ABB RobotStudio station: Escalera.rspag

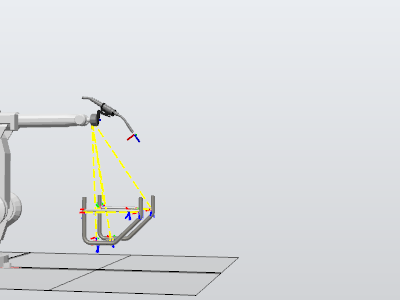
--- station ---
Station Project4 (saved by RobotStudio 23.2.10395.0)
Controller IRB1410_5_144
  mechanical unit ROB_1: IRB1410_5_144__01, 6 joints, base frame (0, 0, 0) mm
Layout (positions relative to the parent item):
  - IRB1410_5_144__01 [mechanism, from %ABB.RobotStudio.Models.IRB1410%\IRB1410_5_144_G_01.rslib] at (0, 0, 0) mm; joint values [0, 0, 0, 0, 0, 0] (rad or m)
  - AW_Gun_PSF_25 [mechanism, from %ABB.RobotStudio.Models.ArcWelding%\AW_Gun_PSF_25.rslib] at (955, 0, 1195) mm, rotated rx 0 ry 90 rz 0 deg
  - escalera [graphiccomponentgroup] at (1200, -200, 400) mm, rotated rx -90 ry 0 rz 0 deg
    - patasescalera:1 [part] at (-235.15, -185.03, 0) mm, size 475.4 x 362.7 x 25.4 mm
    - tubolargo:1 [part] at (-229.58, -85.03, -0.64) mm, rotated rx 90 ry 0 rz 0 deg, size 440 x 19 x 19 mm
    - patasescalera:2 [part] at (-235.69, -185.03, 370) mm, size 475.4 x 362.7 x 25.4 mm
    - tubolargo:2 [part] at (-231.19, -85.03, 370) mm, rotated rx 90 ry 0 rz 0 deg, size 440 x 19 x 19 mm
    - tubo peque\X\F1o:1 [part] at (123.63, -81.8, 370.84) mm, rotated rx -90 ry 89.5 rz -90 deg, size 370 x 19 x 19 mm
    - tubo peque\X\F1o:2 [part] at (-121.37, 167.61, 371.49) mm, rotated rx -90 ry 89.59 rz -90 deg, size 370 x 19 x 19 mm
Attachment: AW_Gun_PSF_25 is attached to IRB1410_5_144__01 / Link6
Targets, tools, work objects and paths stored in the station and not in the controller backup, written as RAPID:
! task T_ROB1
MODULE CalibData
  PERS tooldata AW_Gun:=[TRUE,[[119.5,0,352],[0.890213743,0,0.455543074,0]],[1,[0,0,100],[1,0,0,0],0,0,0]];
  TASK PERS wobjdata Workobject_1:=[FALSE,TRUE,"",[[0,0,0],[1,0,0,0]],[[0,0,0],[1,0,0,0]]];
ENDMODULE

! task T_ROB1
MODULE Module1
  CONST jointtarget Home:=[[0,0,0,0,0,0],[9E+09,9E+09,9E+09,9E+09,9E+09,9E+09]];
  CONST robtarget Mitad1:=[[976.781186414,170.702276534,494.530253281],[0.305176705,0.666129903,-0.637918703,-0.237060876],[-1,0,-1,0],[9E+09,9E+09,9E+09,9E+09,9E+09,9E+09]];
  CONST robtarget Inicio1:=[[972.88593197,180.494399691,477.051816875],[0.385830495,0.691371329,-0.592631267,-0.148083408],[-1,0,-1,0],[9E+09,9E+09,9E+09,9E+09,9E+09,9E+09]];
  CONST robtarget Fin1:=[[973.255,150,480],[0.037823374,0.524703407,-0.706148979,-0.473929685],[-1,0,-2,0],[9E+09,9E+09,9E+09,9E+09,9E+09,9E+09]];
  CONST robtarget Mitad2:=[[978.420658892,-200.453702036,494.554289293],[0.153565718,0.360544064,-0.853445443,-0.343593399],[-1,0,-1,0],[9E+09,9E+09,9E+09,9E+09,9E+09,9E+09]];
  CONST robtarget Fin2:=[[978.421,-220,470],[0.156146418,0.366952713,-0.850711042,-0.342424773],[-1,0,-1,0],[9E+09,9E+09,9E+09,9E+09,9E+09,9E+09]];
  CONST robtarget Inicio2:=[[978.421,-180,470],[0.158675671,0.365866136,-0.848327112,-0.348288837],[-1,0,-1,0],[9E+09,9E+09,9E+09,9E+09,9E+09,9E+09]];
  CONST robtarget Inicio3:=[[1400,-212.929,477.071],[0.120590477,-0.049950211,0.915975615,0.379409523],[-1,-1,1,0],[9E+09,9E+09,9E+09,9E+09,9E+09,9E+09]];
  CONST robtarget Mitad3:=[[1400,-200,490],[0.130526192,0,0.991444861,0],[-1,-1,0,0],[9E+09,9E+09,9E+09,9E+09,9E+09,9E+09]];
  CONST robtarget Fin3:=[[1400,-187.071,477.071],[0.120590477,0.049950211,0.915975615,-0.379409523],[0,0,-1,0],[9E+09,9E+09,9E+09,9E+09,9E+09,9E+09]];
  CONST robtarget Inicio4:=[[1333.134,-191.144,484.911],[0.254887002,0.044943456,-0.951251243,0.167731259],[-1,0,-1,0],[9E+09,9E+09,9E+09,9E+09,9E+09,9E+09]];
  CONST robtarget Mitad4:=[[1323,-191.144,484.911],[0,0,1,0],[-1,0,-1,0],[9E+09,9E+09,9E+09,9E+09,9E+09,9E+09]];
  CONST robtarget Fin4:=[[1313,-191.144,484.911],[0.130526192,0,0.991444861,0],[-1,1,-2,0],[9E+09,9E+09,9E+09,9E+09,9E+09,9E+09]];
  CONST robtarget Inicio5:=[[1313,153.856,484.911],[0.130526192,0,0.991444861,0],[0,0,-1,0],[9E+09,9E+09,9E+09,9E+09,9E+09,9E+09]];
  CONST robtarget Mitad5:=[[1323,160,484.911],[0,0,1,0],[0,1,-2,0],[9E+09,9E+09,9E+09,9E+09,9E+09,9E+09]];
  CONST robtarget Fin5:=[[1333,153.856,480],[0,0,1,0],[0,1,-2,0],[9E+09,9E+09,9E+09,9E+09,9E+09,9E+09]];
  CONST robtarget Inicio6:=[[1405,157.392,476.464],[0.128543206,-0.022665635,0.976382586,0.172162593],[-1,-1,1,0],[9E+09,9E+09,9E+09,9E+09,9E+09,9E+09]];
  CONST robtarget Mitad6:=[[1400,175,485],[0.130526192,0,0.991444861,0],[0,0,-1,0],[9E+09,9E+09,9E+09,9E+09,9E+09,9E+09]];
  CONST robtarget Fin6:=[[1405,178,476.464],[0,0,0.923879533,-0.382683432],[0,1,-2,0],[9E+09,9E+09,9E+09,9E+09,9E+09,9E+09]];
  CONST robtarget Inicio_Ac:=[[1000,180.494,500],[0.38583142,0.69137232,-0.592628496,-0.148087464],[0,0,-1,0],[9E+09,9E+09,9E+09,9E+09,9E+09,9E+09]];
  CONST robtarget M1:=[[1078.634,-187.76,244.444],[0,0,0.984807753,-0.173648178],[-1,0,-1,0],[9E+09,9E+09,9E+09,9E+09,9E+09,9E+09]];
  CONST robtarget I1:=[[1065,-187.76,230],[0.128543206,0.022665635,0.976382586,-0.172162593],[-1,0,-1,0],[9E+09,9E+09,9E+09,9E+09,9E+09,9E+09]];
  CONST robtarget F1:=[[1085,-187.76,230],[0.128543206,0.022665635,-0.976382586,0.172162593],[-1,1,-2,0],[9E+09,9E+09,9E+09,9E+09,9E+09,9E+09]];
  CONST robtarget M2:=[[1078.634,160,242.305],[0.128543206,-0.022665635,-0.976382586,-0.172162593],[0,-2,1,0],[9E+09,9E+09,9E+09,9E+09,9E+09,9E+09]];
  CONST robtarget I2:=[[1090,160,230],[0.128543206,-0.022665635,-0.976382586,-0.172162593],[0,-2,1,0],[9E+09,9E+09,9E+09,9E+09,9E+09,9E+09]];
  CONST robtarget F2:=[[1065,160,225],[0.128543206,-0.022665635,0.976382586,0.172162593],[0,-1,0,0],[9E+09,9E+09,9E+09,9E+09,9E+09,9E+09]];
  CONST robtarget I_Ac:=[[1052.839482654,-170.658992876,275.383668574],[0.128543206,0.022665635,0.976382586,-0.172162593],[-1,0,-1,0],[9E+09,9E+09,9E+09,9E+09,9E+09,9E+09]];
  PROC TubosSuperiores()
    MoveAbsJ Home,v300,z100,AW_Gun\WObj:=wobj0;
    MoveJ Inicio_Ac,v300,z100,AW_Gun\WObj:=wobj0;
    MoveJ Inicio1,v300,z100,AW_Gun\WObj:=wobj0;
    MoveL Mitad1,v300,z100,AW_Gun\WObj:=wobj0;
    MoveL Fin1,v300,z100,AW_Gun\WObj:=wobj0;
    MoveL Inicio2,v300,z100,AW_Gun\WObj:=wobj0;
    MoveL Mitad2,v300,z100,AW_Gun\WObj:=wobj0;
    MoveL Fin2,v300,z100,AW_Gun\WObj:=wobj0;
    MoveJ Inicio3,v300,z100,AW_Gun\WObj:=wobj0;
    MoveL Mitad3,v300,z100,AW_Gun\WObj:=wobj0;
    MoveL Fin3,v300,z100,AW_Gun\WObj:=wobj0;
    MoveJ Inicio4,v300,z100,AW_Gun\WObj:=wobj0;
    MoveL Mitad4,v300,z100,AW_Gun\WObj:=wobj0;
    MoveL Fin4,v300,z100,AW_Gun\WObj:=wobj0;
    MoveJ Inicio5,v300,z100,AW_Gun\WObj:=wobj0;
    MoveL Mitad5,v300,z100,AW_Gun\WObj:=wobj0;
    MoveL Fin5,v300,z100,AW_Gun\WObj:=wobj0;
    MoveJ Inicio6,v300,z100,AW_Gun\WObj:=wobj0;
    MoveL Mitad6,v300,z100,AW_Gun\WObj:=wobj0;
    MoveL Fin6,v300,z100,AW_Gun\WObj:=wobj0;
    MoveAbsJ Home,v300,z100,AW_Gun\WObj:=wobj0;
  ENDPROC
  PROC TuboInferior()
    MoveAbsJ Home,v300,z100,AW_Gun\WObj:=Workobject_1;
    MoveJ I_Ac,v300,z100,AW_Gun\WObj:=Workobject_1;
    MoveL I1,v300,z100,AW_Gun\WObj:=Workobject_1;
    MoveL M1,v300,z100,AW_Gun\WObj:=Workobject_1;
    MoveL F1,v300,z100,AW_Gun\WObj:=Workobject_1;
    MoveJ I2,v300,z100,AW_Gun\WObj:=Workobject_1;
    MoveL M2,v300,z100,AW_Gun\WObj:=Workobject_1;
    MoveL F2,v300,z100,AW_Gun\WObj:=Workobject_1;
    MoveAbsJ Home,v300,z100,AW_Gun\WObj:=Workobject_1;
  ENDPROC
ENDMODULE


--- Controller Data/IRB1410_5_144/RAPID/TASK1/PROGMOD/Module1.mod ---
MODULE Module1
    !***********************************************************
    !
    ! M?dulo:  Module1
    !
    ! Descripción:
    !   <Introduzca la descripción aquí>
    !
    ! Autor: Andrago
    !
    ! Versión: 1.0
    !
    !***********************************************************


    !***********************************************************
    !
    ! Procedimiento Main
    !
    !   Este es el punto de entrada de su programa
    !
    !***********************************************************
    PROC main()
        !Add your code here
    ENDPROC
ENDMODULE
